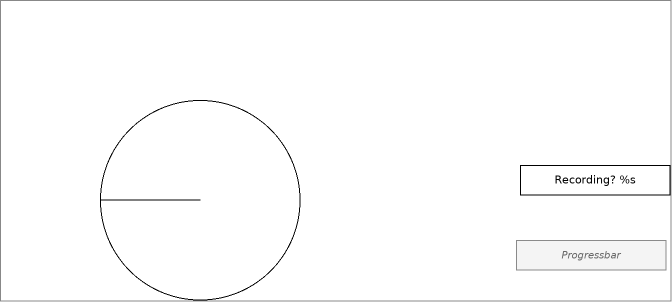
VISUALIZATION Visualization  // 672x302
    Rectangle (520,165 150x30), "Recording? %s", text variable: MAIN.bRecordData
        OnMouseDown: execute { MAIN.bRecordData := NOT MAIN.bRecordData; }
    Ellipse (100,100 200x200)
    Line (200,200) (100,200)
        p2858320360: MAIN.enc_angle
    Progressbar (516,240 150x30), variable: MAIN.cbCurrentBufferLength
END_VISUALIZATION

(* stored: Version 1.1.0.1, ProductVersion 3.1.4022.10
   Visu Visualization: Id {34b664a4-8d8d-4b1d-a719-b54764bdbfc9} *)
